FUNCTION_BLOCK FB_STRING_W (* Converts a STRING to its WSTRING equivalent *)
  (* Standard: 61499-1; Classification: Strings; Function: Conversion; Type: STRING to WSTRING *)
  (* Version 0.0, 2007-08-17, JHC, Holobloc Inc *)
  (* Compiler header: package fb.rt.strings; *)
  (* Compiler classdef: SimpleFB *)
  (* Compiler Java Sun JDK 1.6.0 *)
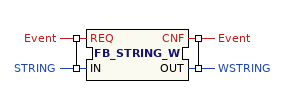
  EVENT_INPUT
    REQ WITH IN; (* Normal Execution Request *)
  END_EVENT
  EVENT_OUTPUT
    CNF WITH OUT; (* Execution Confirmation *)
  END_EVENT
  VAR_INPUT
    IN : STRING;
  END_VAR
  VAR_OUTPUT
    OUT : WSTRING;
  END_VAR
  ALGORITHM REQ IN Java:
OUT.value = new String(IN.value, 0, IN.length);
  END_ALGORITHM
END_FUNCTION_BLOCK
